(* PLC project tni_clock, Dassault Systèmes ControlBuild 2024x *)
(* stored: creationDateTime 2023-10-05T15:44:29-01:00 *)

CONFIGURATION tni_clock
  VAR_GLOBAL
    simuperiod : REAL := 50000.0;
    taskname : STRING(50) := 'tni_clock.exe';
    allowpreconditions : BOOL := true;
    allowpostconditions : BOOL := true;
  END_VAR
END_CONFIGURATION
